TYPE
    ST_CSV_Detail : STRUCT
        DetailID  : UDINT;
        DataCount : UDINT;
        Datas     : ARRAY[1..MAX_DATA_COUNT] OF T_MaxString;
    END_STRUCT
END_TYPE

(* stored: Version 1.1.0.1
   DUT ST_CSV_Detail: Id {9a483490-634f-4104-996e-826265d34d59} *)
